(* CODESYS project mqtt.sharememory.gps.20211124.1.project

Project tree, tasks and I/O mapping:
  Device : Changsha Xiangji-ARM Cortex A9(xilinx zynq7000)-linux, Changsha Xiangji Hiden Technology Co.Ltd, version 3.5.10.40
    application Application
      libraries: Standard, * (System); SysShm, * (System); SysTypes2 Interfaces, * (System); CAA Types Extern, 3.5.13.0 (CAA Technical Workgroup); CAA Net Base Services, 3.5.15.0 (CAA Technical Workgroup); CAA Memory, 3.5.12.0 (CAA Technical Workgroup); SysFile, 3.5.15.0 (System); CAA SerialCom, 3.5.15.0 (CAA Technical Workgroup); MIC7001 base library, 1.11 (Cyber-MI.com); CAA DTUtil Extern, 3.5.12.0 (CAA Technical Workgroup)
      task Task_mqtt (cyclic, interval 200 ms, priority 19) calls prg_mqtt, prg_gps, prg_jt808
      global variables GVL
      data type ret_index
      MQTT_Client/
        Function Blocks/
          function block FB_CalculateRemainingLength [ST]
          function block FB_DecodeRemainingLength [ST]
          function block FB_MQTTClient [ST]: m_fill_subscribe_buf, m_fill_publish_buf, m_fill_connect_buf, rm_return, m_read_config
          function block FB_Random [ST]
        Structs/
          data type DUT_json
        Functions/
          function real_arr2string [ST]
          function MQTTPacket_encode [ST]
          function MQTTPacket_len [ST]
          function MQTT_connect_len [ST]
          function arr2json_model [ST]
          function json2arr [ST]
          function get_sub_string [ST]
          function count_char_in_string [ST]
          function rm_left [ST]
          function real2string [ST]
        program prg_mqtt [CFC]: ACT_boot, ACT_publish, ACT_recv_proc, ACT_first_buffer, ACT_normal_buffer, ACT_running_light, proc_get_command, proc_set_command, find_key
      gps/
        programs/
          program prg_gps [ST]
        Structs/
          data type stShmJT808Down
          data type stLocationExt
          data type stShmJT808Up
          data type stLocationBase
          data type stCanFrm
          data type nmeaTIME
          data type nmeaGPRMC
        functions/
          function nmea_parse_time [ST]
          function nmea_parse_date [ST]
          function get_latlon_from_str [ST]
          function nmea_parse_GPRMC [ST]
          function get_sub_string_1 [ST]
        functionblocks/
          function block Com_gps [ST]
      program prg_jt808 [ST]: send_to_server, read_from_server, init_shm
    SoftMotion General Axis Pool
  text list GlobalTextList
  5ce3da45-db07-42e7-a21c-a00fff4ed8f6|C:\Users\pengriguang\Desktop\cyber-tftp\huanweiche.bmp
*)

// Device/Application/ret_index
{attribute 'qualified_only'}
{attribute 'strict'}
TYPE ret_index :
(
	start := 0,
	cntr_box,
	cntr_lock,
	hours_e,
	fuel_work,
	fuel_idle
);
END_TYPE

// Device/Application/MQTT_Client/Structs/DUT_json
TYPE DUT_json :
STRUCT
	key:STRING(32);
	value_dint : DINT;
	value_real : REAL;
	value_str : STRING(256);
	val_tp : UINT;  //0:  int,   1: real,    2: string
END_STRUCT
END_TYPE

// Device/Application/gps/Structs/stShmJT808Down
TYPE stShmJT808Down :  // JT808下行数据
STRUCT
	location_interval:DINT;  // 位置信息发送间隔， 单位： ms
	ctrl : DINT;   // 车辆控制命令
END_STRUCT
END_TYPE

// Device/Application/gps/Structs/stLocationExt
TYPE stLocationExt :
STRUCT
	km_all: DINT;  // km all
	fuel:INT;   // fuel meter
	speed: INT;  // speed can
	lac:DINT; 
	cid:DINT;
	fuel_trip:DINT; // 本行程油耗
	fuel_all:DINT; 
	fuel_r_h:DINT;  // 0.05L/h
	fuel_r_l:DINT;  //  1/512Km/L
END_STRUCT
END_TYPE

// Device/Application/gps/Structs/stShmJT808Up
TYPE stShmJT808Up :   // 发送到服务器的上行数据
STRUCT
    location:stLocationBase;
	loc_ext:stLocationExt;
	can_data:stCanFrm;
END_STRUCT
END_TYPE

// Device/Application/gps/Structs/stLocationBase
TYPE stLocationBase :
STRUCT
	warning : UDINT;
    status : UDINT;
    latitude : DINT;
    longitude : DINT;
    altitude : INT;
    speed : INT;
    bearing : INT;
    asc_time :ARRAY[0..5] OF BYTE;  // ascii YYMMDDhhmmss (GMT+8)
END_STRUCT
END_TYPE

// Device/Application/gps/Structs/stCanFrm
TYPE stCanFrm :
STRUCT
	sn:UDINT;  // 每次更新内容后加一，用于通知底层发送程序
	id:UDINT;  //  CAN id
	data:ARRAY[0..7] OF BYTE;  // 8个字节 数据
END_STRUCT
END_TYPE

// Device/Application/gps/Structs/nmeaTIME
TYPE nmeaTIME :
STRUCT
	year:DINT;
	month:DINT;
	day:DINT;
	hour:DINT;
	minute:DINT;
	second:DINT;
	hsecond:DINT;
END_STRUCT
END_TYPE

// Device/Application/gps/Structs/nmeaGPRMC
TYPE nmeaGPRMC :
STRUCT
	utc : nmeaTIME;
	status : STRING(1);
	lat : REAL;
	ns : STRING(1);
	lon : REAL;
	ew : STRING(1);
	speed : REAL;
	direction : REAL;
	declination : REAL;
	declin_ew : STRING(1);
	mode : STRING(1);
END_STRUCT
END_TYPE

// Device/Application/GVL
{attribute 'qualified_only'}
VAR_GLOBAL PERSISTENT RETAIN
	ret_val1: DINT;  
	ret_val2: Dint;
END_VAR

VAR_GLOBAL CONSTANT
	TYPE_DINT:UINT := 0;
	TYPE_REAL:UINT := 1;
	TYPE_STRING:UINT := 2;
END_VAR

VAR_GLOBAL
	mqtt_interval : DINT := 5;  //mqtt package interval of publish to server
END_VAR

// Device/Application/MQTT_Client/prg_mqtt
PROGRAM prg_mqtt
VAR_INPUT
	mode_set :DINT := 99;
END_VAR
VAR
	FB_MQTTClient_0: FB_MQTTClient;
	
	//topic : STRING(255) := '/sys/a1SB8J9cA4L/CMI010319120011/thing/model/up_raw';
	//topic : STRING(255) := '/a1SB8J9cA4L/CMI010319120011/user/to_app';
	payload : STRING(255) := '{"RPM": 1234, "Hours": 2345}';
	
	//subscribe : STRING(255) := '/a1SB8J9cA4L/CMI010319120011/user/from_app';
	
	xPub : BOOL := FALSE;
	xSub : BOOL := FALSE;
	xBooted :BOOL := FALSE;
	
	ton_pub : ton;
	
	val_payload:ARRAY[0..32] OF dut_json;
	rpm_value : DINT := 1000;
	hours_value :REAL := 680;
	time_value : STRING;
	sn_value : STRING(128);
	lac_str:STRING(128);
	cid_str:STRING(128);
	press_value :REAL := 20.1;
	
	recv_data : ARRAY[0..32] OF DUT_json;
	old_recv_cntr:UDINT := 0;
	payload_len :INT;
	
	mqtt_first :BOOL := TRUE;
	ton_running:ton:=(pt := T#500MS);
	led_run:BOOL := FALSE;
	led_err:BOOL := FALSE;
	led_usr:BOOL := FALSE;
	pkg_id :DINT := 0;
	i :DINT;
	hour_today:REAL := 2.0;
	pub_cntr :DINT := 0;
	
	press:DWORD;
	oil :DWORD;
	temp : DWORD;
	send_serial:DINT := 0;  // 发送帧的序列号
	arr : ARRAY [0..19] OF REAL;
	
	angle:REAL := 60.0;
	length:REAL := 0.0;
END_VAR

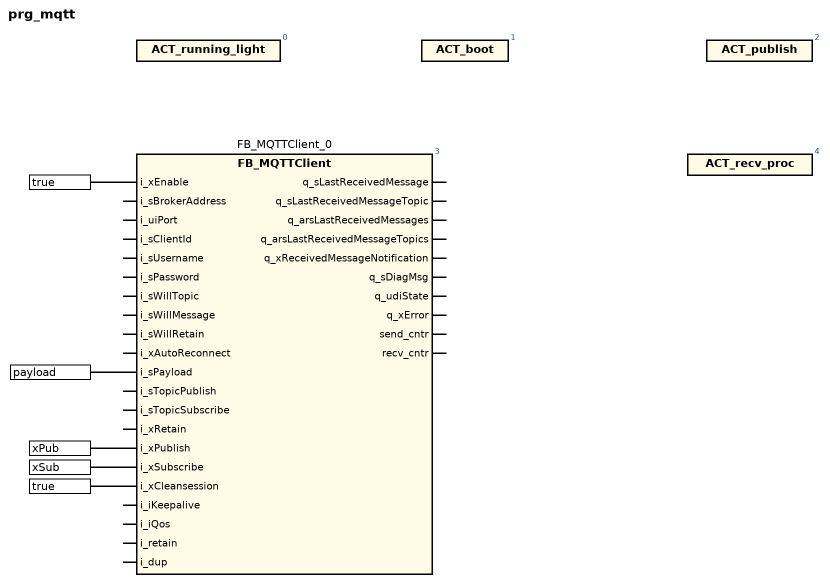
ACT_running_light();
ACT_boot();
ACT_publish();
FB_MQTTClient_0(
    i_xEnable := true,
    i_sPayload := payload,
    i_xPublish := xPub,
    i_xSubscribe := xSub,
    i_xCleansession := true); // FB_MQTTClient
ACT_recv_proc();

ACTION ACT_boot:
IF NOT xbooted THEN
	IF FB_MQTTClient_0.q_udiState = 60 THEN
		FB_MQTTClient_0.i_xSubscribe := TRUE;
		xBooted := TRUE;
	END_IF
END_IF
END_ACTION

ACTION ACT_publish:
IF FB_MQTTClient_0.q_udiState <> 60 THEN   //not ready, return and wait
	xPub := FALSE;
	RETURN;
END_IF

IF mqtt_first THEN
	mqtt_first := FALSE;
	ACT_first_buffer();
	xPub := TRUE;
	RETURN;
END_IF

ton_pub(in := NOT ton_pub.Q, pt := ANY_TO_TIME(gvl.mqtt_interval*1000));   // second to ms
IF ton_pub.Q THEN
	ACT_normal_buffer();
	xPub := TRUE;
ELSE
	xPub := FALSE;
END_IF
END_ACTION

ACTION ACT_recv_proc:
(*
	cmd:  	set, get          			//命令字, set:设置参数或者执行命令，  get：点播数据或参数
	act:  	lock, unlock, reboot		//动作类型
	grade:  1, 2, 3, 4					//动作级别
	delay:  0, 60, 3600					//延迟时间,单位： 秒
*)

IF old_recv_cntr = FB_MQTTClient_0.recv_cntr THEN  //no new message
	RETURN;
END_IF
old_recv_cntr := FB_MQTTClient_0.recv_cntr;

payload_len := json2arr(json := FB_MQTTClient_0.q_sLastReceivedMessage, pArr := ADR(recv_data), max_len := 32);
IF payload_len = 0 THEN
	RETURN;
END_IF

i := find_key(key := 'cmd');
IF i >= 0 AND recv_data[i].val_tp = GVL.TYPE_STRING THEN 
	IF  recv_data[i].value_str = 'get' THEN
		proc_get_command();
	ELSIF recv_data[i].value_str = 'set' THEN
		proc_set_command();
	END_IF
END_IF
END_ACTION

ACTION ACT_first_buffer:

val_payload[0].key := 'sn';
val_payload[0].val_tp := GVL.TYPE_STRING;
IF MIC7001_base.read_sn(ADR(sn_value)) THEN
	val_payload[0].value_str := sn_value;
ELSE
	val_payload[0].value_str := 'SN Error';
END_IF

val_payload[1].key := 'lac';
val_payload[1].val_tp := GVL.TYPE_STRING;

val_payload[2].key := 'cid';
val_payload[2].val_tp := GVL.TYPE_STRING;

IF MIC7001_base.read_location(lac := ADR(lac_str), ci := ADR(cid_str)) THEN
	val_payload[1].value_str := lac_str; 
	val_payload[2].value_str := cid_str; 
ELSE
	val_payload[1].value_str := 'lac_error'; 
	val_payload[2].value_str := 'cid_error'; 
END_IF

payload := arr2json_model(arr := val_payload, num := 3);
END_ACTION

ACTION ACT_normal_buffer:
// 数据太多，分帧发送  0~3 共4帧， 可以把需要同时发送的关联数据放在一帧中
CASE send_serial OF
0:	
	val_payload[0].key := 'BoxNo';
	val_payload[0].val_tp := GVL.TYPE_STRING; 
	val_payload[0].value_str := 'Box123456'; 

	val_payload[1].key := 'digi_0_29';
	val_payload[1].val_tp := GVL.TYPE_DINT; 
	val_payload[1].value_dint.0 := TRUE; //bForward;   // 前进档
	val_payload[1].value_dint.1 := FALSE; //bBackward;   // 前进档
	// ...
	val_payload[1].value_dint.29 := TRUE;  // bLocked;   // 属具已闭锁
	
	
	val_payload[2].key := 'digi_30_59';
	val_payload[2].val_tp := GVL.TYPE_DINT; 
	val_payload[2].value_dint := 12345;

	val_payload[3].key := 'digi_60_89';
	val_payload[3].val_tp := GVL.TYPE_DINT; 
	val_payload[3].value_dint := 12345; 

	val_payload[4].key := 'digi_90_119';
	val_payload[4].val_tp := GVL.TYPE_DINT; 
	val_payload[4].value_dint := 12345;  	
(*  ana_0_19	
0 发动机转速
1 发动机水温
2 发动机机油压力
3 发动机燃油箱体积
4 变速箱涡轮转速
5 变速箱温度
6 变速箱压力
7 吊载重量
8 前伸距
9 臂架角度
10 臂架长度
11 刹车油温度
12 液压油温度
13 俯仰动作手柄输入
14 伸缩动作手柄输入
15 吊具旋转动作输入
16 吊具侧移动作输入
17 整机故障代码
*)
	val_payload[5].key := 'ana_0_19';
	val_payload[5].val_tp := GVL.TYPE_STRING;
    arr[0] := 123; // gvl.rpm;
    arr[1] := 345.5678; // gvl.temp;
    arr[2] := 888; // gvl.press;t
	
	arr[8] := 4.2;   // 前伸距离 
	arr[9] := angle;   // 臂架角度
	arr[10] := length;   // 臂架长度
	
	angle := 60;
	
	length := length + 0.3;
	IF length > 7.2 THEN
		length := 0;
	END_IF
	
	// ...
    arr[17] := 16#01020304; // gvl.errorcode
	val_payload[5].value_str := real_arr2string(arr, 18); 
	
	payload := arr2json_model(arr := val_payload, num := 6);
	
1:
	val_payload[0].key := 'BoxNo';
	val_payload[0].val_tp := GVL.TYPE_STRING; 
	val_payload[0].value_str := 'Box123456'; 

	val_payload[1].key := 'digi_0_29';
	val_payload[1].val_tp := GVL.TYPE_DINT; 
	val_payload[1].value_dint := 12345; 
	
	val_payload[2].key := 'digi_30_59';
	val_payload[2].val_tp := GVL.TYPE_DINT; 
	val_payload[2].value_dint := 12345;

	val_payload[3].key := 'digi_60_89';
	val_payload[3].val_tp := GVL.TYPE_DINT; 
	val_payload[3].value_dint := 12345; 

	val_payload[4].key := 'digi_90_119';
	val_payload[4].val_tp := GVL.TYPE_DINT; 
	val_payload[4].value_dint := 12345;  
(*  ana_20_39
0 吊箱总数
1 旋锁计数
2 伸出PWM值
3 缩回PWM值
4 仰起PWM值
5 俯下PWM值
6 正面吊左无杆腔压力
7 正面吊右有杆腔压力
8 正面吊右无杆腔压力
9 正面吊伸缩压力
10 设备行驶速度
11 液压系统压力
12 力矩百分比
*)	
	val_payload[5].key := 'ana_20_39';
	val_payload[5].val_tp := GVL.TYPE_STRING;
    arr[0] := 333; // gvl.box_all;
    arr[1] := 555; // gvl.lock_all;
    arr[2] := 1357; // gvl.pwm_out;
	// ...
    arr[12] := 82; // gvl.tor
	val_payload[5].value_str := real_arr2string(arr, 13); 
	
	payload := arr2json_model(arr := val_payload, num := 6);
2:
	val_payload[0].key := 'BoxNo';
	val_payload[0].val_tp := GVL.TYPE_STRING; 
	val_payload[0].value_str := 'Box123456'; 

	val_payload[1].key := 'digi_0_29';
	val_payload[1].val_tp := GVL.TYPE_DINT; 
	val_payload[1].value_dint := 12345; 
	
	val_payload[2].key := 'digi_30_59';
	val_payload[2].val_tp := GVL.TYPE_DINT; 
	val_payload[2].value_dint := 12345;

	val_payload[3].key := 'digi_60_89';
	val_payload[3].val_tp := GVL.TYPE_DINT; 
	val_payload[3].value_dint := 12345; 

	val_payload[4].key := 'digi_90_119';
	val_payload[4].val_tp := GVL.TYPE_DINT; 
	val_payload[4].value_dint := 12345;  
(*  ana_40_59
0 发动机运行时间
1 发动机故障SPN码
2 发动机后处理SPN码
3 发动机蓄电池电压
4 总油耗
5 工作油耗
6 怠速油耗
7 发动机瞬时油耗
8 发动机怠速工作时长
9 刹车踏板制动百分比
10 油门踏板百分比
11 变速箱SPN_L
12 变速箱SPN_H
13 左前轮胎外侧胎压
14 左前轮胎内侧胎压
15 右前轮胎外侧胎压
16 右前轮胎内侧胎压
17 左后轮胎胎压
18 右后轮胎胎压
*)	
	val_payload[5].key := 'ana_40_59';
	val_payload[5].val_tp := GVL.TYPE_STRING;
    arr[0] := 333; // 
    arr[1] := 555; // 
    arr[2] := 1357; // 
	arr[3] := 28.1;
	arr[4] := 12345.6;
	arr[5] := 10000;
	arr[6] := 2345.6;
	arr[7] := 2.6;
	// ...
	arr[17] := 2.7;
	arr[18] := 2.9;
	val_payload[5].value_str := real_arr2string(arr, 19); 
	
	payload := arr2json_model(arr := val_payload, num := 6);

3:
	val_payload[0].key := 'BoxNo';
	val_payload[0].val_tp := GVL.TYPE_STRING; 
	val_payload[0].value_str := 'Box123456'; 

	val_payload[1].key := 'digi_0_29';
	val_payload[1].val_tp := GVL.TYPE_DINT; 
	val_payload[1].value_dint := 12345; 
	
	val_payload[2].key := 'digi_30_59';
	val_payload[2].val_tp := GVL.TYPE_DINT; 
	val_payload[2].value_dint := 12345;

	val_payload[3].key := 'digi_60_89';
	val_payload[3].val_tp := GVL.TYPE_DINT; 
	val_payload[3].value_dint := 12345; 

	val_payload[4].key := 'digi_90_119';
	val_payload[4].val_tp := GVL.TYPE_DINT; 
	val_payload[4].value_dint := 12345;  
(*  ana_20_39
设备类型
生产年份
车号
设备品牌
发动机类型
变速箱类型
驱动桥类型
吊具类型
吊具程序版本号
主机程序版本号
吊重箱数量
*)	
	val_payload[5].key := 'ana_60_79';
	val_payload[5].val_tp := GVL.TYPE_STRING;
    arr[0] := 333; // gvl.
    arr[1] := 555; // gvl.
    arr[2] := 1357; // gvl.
	// ...
    arr[10] := 82; // gvl.
	val_payload[5].value_str := real_arr2string(arr, 11); 
	
	payload := arr2json_model(arr := val_payload, num := 6);
4:
	val_payload[0].key := 'BoxNo';
	val_payload[0].val_tp := GVL.TYPE_STRING; 
	val_payload[0].value_str := 'Box123456'; 

	val_payload[1].key := 'digi_0_29';
	val_payload[1].val_tp := GVL.TYPE_DINT; 
	val_payload[1].value_dint := 12345; 
	
	val_payload[2].key := 'digi_30_59';
	val_payload[2].val_tp := GVL.TYPE_DINT; 
	val_payload[2].value_dint := 12345;

	val_payload[3].key := 'digi_60_89';
	val_payload[3].val_tp := GVL.TYPE_DINT; 
	val_payload[3].value_dint := 12345; 

	val_payload[4].key := 'digi_90_119';
	val_payload[4].val_tp := GVL.TYPE_DINT; 
	val_payload[4].value_dint := 12345;  
	
(*  ana_80_99
锂电池SOC
。。。
。。。
*)	
	val_payload[5].key := 'ana_80_99';
	val_payload[5].val_tp := GVL.TYPE_STRING;
    arr[0] := 333; // gvl.
    arr[1] := 555; // gvl.
    arr[2] := 1357; // gvl.
	// ...
    arr[10] := 82; // gvl.
    arr[11] := 12; // gvl.
	
IF prg_gps.packGPRMC.status = 'A' THEN  // GPS定位成功
	arr[12] := prg_gps.packGPRMC.lat*1000000;    //维度 * 1000000
	arr[13] := prg_gps.packGPRMC.lon*1000000;	 //经度 * 1000000
END_IF
	val_payload[5].value_str := real_arr2string(arr, 14);
	
	payload := arr2json_model(arr := val_payload, num := 6);	
	
END_CASE


send_serial := send_serial + 1;
IF send_serial > 4 THEN
	send_serial := 0;
END_IF
END_ACTION

ACTION ACT_running_light:
ton_running(in := NOT ton_running.Q);
IF ton_running.Q THEN
	led_run := NOT led_run;
	led_usr := FALSE;
END_IF

IF FB_MQTTClient_0.q_udiState <> 60 THEN
	led_usr := TRUE;
END_IF
END_ACTION

ACTION proc_get_command:
(*
	cmd:  	get  	//命令字, get：点播数据或参数
	rpm:  	15		//点播转速， 上传15次
	press:  0		//点播压力， 持续上传
	fuel_all: 1	  	//点播总油耗，上传一次 					
*)
END_ACTION

ACTION proc_set_command:
(*
	cmd:  	set  	          	//命令字, set:设置参数或者执行命令，  get：点播数据或参数
	interval:	15				//设置上传间隔： 15秒
	act:  	lock, unlock		//锁机动作类型
	grade:  1, 2, 3, 4			//动作级别
	delay:  0, 60, 3600			//延迟时间,单位： 秒
*)

// check lock command 
i := find_key(key := 'act');
IF i >= 0 AND recv_data[i].val_tp = GVL.TYPE_STRING  THEN
  //
END_IF
END_ACTION

METHOD find_key : dint
VAR_INPUT
	key :STRING(32);
END_VAR
VAR
	i :UINT;
END_VAR
find_key := -1;

FOR i := 0 TO payload_len-1 DO
	IF key = recv_data[i].key THEN
		find_key := i;
		RETURN;
	END_IF
END_FOR

RETURN; // not find,  return -1
END_METHOD

END_PROGRAM

// Device/Application/MQTT_Client/Function Blocks/FB_MQTTClient
(*  mqtt client for MIC7001
    by zhoujihui@gmail.com
*)
FUNCTION_BLOCK FB_MQTTClient
VAR_INPUT
	// Enables the Function block, The rising Edge of this Input automatically connects to the MQTT Broker - Standard: TRUE
	i_xEnable: BOOL := TRUE;
	// IP-Address (example: 192.168.178.101) or Webaddress (www.mqtt-dashboard.com) of the MQTT-Broker
	i_sBrokerAddress: STRING(255) := '47.107.240.29';
	// Port of the MQTT-Broker - Standard: 1883
	i_uiPort: UINT := 1883;
	// clientId
	i_sClientId: STRING(255) := 'MIC7001 client Id';
	// Optional Username if required
	i_sUsername: STRING(255) := '';
	// Optional Password if required
	i_sPassword: STRING(255) := '';
	// Last Will Topic if required (Automatically enables Will Message if changed) - otherwise leave untouched
	i_sWillTopic: STRING(255) := '';
	// Last Will Message if required - otherwise leave untouched
	i_sWillMessage: STRING(255) := '';
	// Retain Last Will Message, if required Standard: FALSE - otherwise leave untouched 
	i_sWillRetain: BOOL := FALSE;	
	// Automatically try to reconnect after an Exception - Standard: TRUE
	i_xAutoReconnect: BOOL := TRUE;
	// PayLoad to Publish
	i_sPayload: STRING(255) := '';
	// Topic to Publish to
	i_sTopicPublish: STRING(255) := '/MIC7001/without/config/files';
	// Topic to Subscribe
	i_sTopicSubscribe: STRING(255) := '';
	// Retain Flag Forces the Broker to Retain the Last Mesage - Standard: TRUE
	i_xRetain: BOOL := TRUE;
	// Publish the Payload to the Topic of the MQTT-Broker
	i_xPublish: BOOL:=FALSE;
	// Subscribe to the Topic given to the Input i_sTopicSubscribe
	i_xSubscribe: BOOL:=FALSE;
	// clean session
	i_xCleansession : BOOL := FALSE;
	// keep alive
	i_iKeepalive :INT := 60000;
	// QoS of publish packet
	i_iQos : BYTE := 0;
	// retain
	i_retain : BOOL := FALSE;
	// dup
	i_dup :BOOL := FALSE;
	
END_VAR
VAR_OUTPUT
	// Message Received from a subsribed Topic
	q_sLastReceivedMessage: STRING(255);
	// Topic Message Received
	q_sLastReceivedMessageTopic: STRING(255);	
	// Last 25 Received Messages
	q_arsLastReceivedMessages: STRING(255);
	// Last 25 Topics Received
	q_arsLastReceivedMessageTopics: STRING(255);	
	// Message Received Notification
	q_xReceivedMessageNotification: BOOL;
	// Diag Message
	q_sDiagMsg: STRING(255);
	// Current State of the Function Block
	q_udiState: UDINT;
	// Error Flag
	q_xError: BOOL;
	//publish message counter
	send_cntr :UDINT := 0;
	//received message counter
	recv_cntr: UDINT := 0;
END_VAR
VAR
	R_TRIG_Enable: R_TRIG;

	diResult: CAA.SIZE;
	IFB_CalculateRemainingLength: FB_CalculateRemainingLength;
	IFB_Random: ARRAY[0..9] OF FB_Random;
	wKeepAlive: WORD := 0;
	IoCtlParameter : DINT := 1;

	R_TRIG_Publish: R_TRIG;
	R_TRIG_Subscribe: R_TRIG;

	uiYear:UINT;
	uiMonth: UINT;
	uiDay: UINT;
	uiHour: UINT;
	uiMinute: UINT;
	uiSecond: UINT;
	
	TON_TimeOut: ton;
	wTimeOutValue: WORD;
	udiLastState: UDINT;
	
	xResultDisconnect: BOOL;
	QI: INT;
	
	iIndexCount: INT;
	wPacketIdentifierCount: WORD :=0;
	uiPayLoadLength: uint;
	
	xPublish: BOOL;
	xSubscribe: BOOL;
	
	i: INT;

	hSock:RTS_IEC_HANDLE;
	pSock_create_rst: POINTER TO RTS_IEC_RESULT;
	pSock_recv_rst: POINTER TO RTS_IEC_RESULT;
	pSock_send_rst: POINTER TO RTS_IEC_RESULT;

	ui_rc_disconnect : UDINT;
	pInaddr:POINTER TO STRING;
	
	tcp_client : NBS.TCP_Client;
	tcp_connection : CAA.HANDLE;
	tcp_send : NBS.TCP_Write;
	tcp_recv : NBS.TCP_Read;
	s_send_buf : ARRAY[0..999] OF BYTE;
	s_recv_buf : ARRAY[0..999] OF BYTE;
	udi_time_out : UDINT;
	server_ip : NBS.IP_ADDR;
	buf_size : CAA.size;
	recv_len : INT;

	header :BYTE ; 
	bytes_len_rem : INT;
	length_topic : INT;
	recv_qos : BYTE := 0;
	id_msb : BYTE;
	id_lsb : BYTE;
	hFile: RTS_IEC_HANDLE;
	udiOpenError: RTS_IEC_RESULT;
	udiReadError: RTS_IEC_RESULT;
	str_size: __XWORD;
	udiByteRead: LWORD;	
	str_temp:STRING(255);
	error_cntr : DINT := 0;
END_VAR


R_TRIG_Enable(CLK:=i_xEnable);
R_TRIG_Publish(CLK:=i_xPublish);
R_TRIG_Subscribe(CLK:=i_xSubscribe);

IF (R_TRIG_Publish.Q) THEN
	xPublish:=TRUE;
END_IF

IF (R_TRIG_Subscribe.Q) THEN
	xSubscribe:=TRUE;
END_IF

CASE q_udiState OF
//0: Wait for Enable
0: 	wTimeOutValue:=0;
	
	IF (NOT q_xError) THEN	
		q_sDiagMsg:='Wait for Enable';
	END_IF
	
	IF (i_xEnable OR (i_xAutoReconnect AND q_xError)) THEN
		IF m_read_config() THEN
			q_xError := FALSE;
			q_udiState:=5;
			tcp_client(xEnable := FALSE);
			server_ip.sAddr := i_sBrokerAddress;
			tcp_client.xEnable := TRUE;			
			q_sDiagMsg:='Creating TCP connect';
		ELSE
			q_xError := TRUE;
			q_sDiagMsg:='Failed reading config files';
			q_udiState:=99;
		END_IF
		
	END_IF

5:  
	IF tcp_client.xActive THEN
		q_udiState := 15;
		q_sDiagMsg:='Initialize send-Buffer';
	END_IF
	
	wTimeOutValue:=3000;
	IF (TON_TimeOut.Q) THEN
		q_udiState:=0;	
	END_IF		

//15: Initialize OutBuffer
15:
	buf_size := m_fill_connect_buf();
	IF buf_size > 0 THEN
		tcp_send.szSize := buf_size; 
		tcp_send(xExecute := FALSE);
		tcp_send.xExecute := TRUE;
		tcp_recv.xEnable := TRUE;
		
		q_udiState:=20;
		q_sDiagMsg:='Connect to MQTT-Broker';
	ELSE
		q_xError := TRUE;
		q_sDiagMsg:='Send buffer is Error.';
		q_udiState:=0;
	END_IF
	
//20: Send Connect	
20:		
	wTimeOutValue:=1000;
	tcp_recv(hConnection := tcp_connection, szSize := 1024, pData := ADR(s_recv_buf));
	IF tcp_recv.xReady  THEN
		q_udiState:= 30;
	END_IF
	
	IF (TON_TimeOut.Q) THEN
		q_udiState:=0;	
		q_xError := TRUE;
		q_sDiagMsg:='Connecting to MQTT-Broker (MQTT Control Packet) Timed out';
	END_IF
//30: Analyze CONNACK
30:	q_sDiagMsg:='Analyze connack';
	wTimeOutValue:=0;
	
	IF (s_recv_buf[0] = 32 AND s_recv_buf[3] = 0) THEN
		q_udiState := 60;
	ELSE
		//Return code repsone (2nd Byte): 
		//0: Connection Accepted
		//1: Connection Refused, unacceptable protocol version
		IF (s_recv_buf[3] = 1) THEN
			q_sDiagMsg:='Connection Refused, unacceptable protocol version';
		END_IF
		//2: Connection Refused, identifier rejected
		IF (s_recv_buf[3] = 2) THEN
			q_sDiagMsg:='Connection Refused, identifier rejected';
		END_IF
		//3: Connection Refused, Server unavailable
		IF (s_recv_buf[3] = 3) THEN
			q_sDiagMsg:='Connection Refused, Server unavailable';
		END_IF		
		//4: Connection Refused, bad Username or passworrd
		IF (s_recv_buf[3] = 4) THEN
			q_sDiagMsg:='Connection Refused, bad Username or password';
		END_IF	
		//5: Connection Refused, not autorized
		IF (s_recv_buf[3] = 5) THEN
			q_sDiagMsg:='Connection Refused, not autorized';
		END_IF	
		q_xError := TRUE;
		q_udiState := 90;	
	END_IF
	
//60: Wait for Publish or Disconnect (Enable low)
60:	q_sDiagMsg:='Wait for Publish or Subscribe or Disconnect (Enable low)';
	wTimeOutValue:=0;
	q_xReceivedMessageNotification:= FALSE;

	IF (xPublish) THEN
		xPublish:=FALSE;
		q_udiState := 70;	
	END_IF
	IF (xSubscribe) THEN
		xSubscribe:=FALSE;
		q_udiState := 65;	
	END_IF
	IF (NOT i_xEnable) THEN
		q_udiState := 80;	
	END_IF
	
	tcp_recv(hConnection := tcp_connection, szSize := 1024, pData := ADR(s_recv_buf));
	IF tcp_recv.szCount > 2 THEN
		header := s_recv_buf[0];
		IF header.5 AND header.4 AND tcp_recv.szCount < 1024 THEN   // publish:  0x30
			q_xReceivedMessageNotification:= TRUE;
			diResult := tcp_recv.szCount;
			q_udiState := 63;
			
		END_IF	
	END_IF
	
//Analyze Publish Message from Broker
63: q_sDiagMsg:='Analyze Publish Message from Broker';
	wTimeOutValue:=0;

	IFB_CalculateRemainingLength(wNumberOfBytes:=ANY_TO_WORD(diResult-2));
	bytes_len_rem := IFB_CalculateRemainingLength.iNumberOfBytesRemianingLengthField;
	length_topic := BYTE_TO_INT(s_recv_buf[bytes_len_rem+1])*256 + s_recv_buf[bytes_len_rem+2];
	IF length_topic > 128 THEN
		q_udiState := 60;
		RETURN;	
	END_IF
	
	uiPayLoadLength:=ANY_TO_UINT(diResult - length_topic - 1 - bytes_len_rem - 2);
	header := s_recv_buf[0];
	
	recv_qos := 0;
	IF header.1 OR header.2 THEN //Qos > 0
		uiPayLoadLength :=  uiPayLoadLength - 2;  //remove 2bytes of packet Id
		IF header.1 THEN
			recv_qos := 1;
		ELSIF header.2 THEN
			recv_qos := 2;
		END_IF	

		id_msb := s_recv_buf[1+bytes_len_rem + 2 + length_topic];
		id_lsb := s_recv_buf[1+bytes_len_rem + 2 + length_topic+1];
	END_IF
	
	mem.MemFill(ADR(q_sLastReceivedMessage),255,0);
	mem.MemFill(ADR(q_sLastReceivedMessageTopic),255,0);
	MEM.MemMove(ADR(s_recv_buf[diResult-uiPayLoadLength]),ADR(q_sLastReceivedMessage),uiPayLoadLength);
	MEM.MemMove(ADR(s_recv_buf[IFB_CalculateRemainingLength.iNumberOfBytesRemianingLengthField+3]),ADR(q_sLastReceivedMessageTopic),length_topic);
	
	q_arsLastReceivedMessageTopics:=q_sLastReceivedMessageTopic;
	q_arsLastReceivedMessages:=q_sLastReceivedMessage;
	
	diResult:=0;
	recv_cntr := recv_cntr + 1;
	IF recv_qos = 0 THEN
		q_udiState := 60;
	ELSIF recv_qos = 1 THEN
		
		s_send_buf[0] := 16#40;  //type: puback
		s_send_buf[1] := 2;
		s_send_buf[2] := id_msb;
		s_send_buf[3] := id_lsb;
		tcp_send(xExecute := FALSE);
		tcp_send.xExecute := TRUE;
		tcp_send.szSize := 4;
		q_udiState := 64; // send ack
		wTimeOutValue:=1000;
		q_sDiagMsg:='Send ack to broker';
	ELSE  // qos = 2, not support yet
		q_udiState := 60;
	END_IF	

64:
	IF tcp_send.xDone THEN
		q_udistate := 60;
	END_IF
//65: Subscribe to Topic
65: q_sDiagMsg:='Subscribe to Topic';
	wTimeOutValue:=1000;
	
	buf_size := m_fill_subscribe_buf();
	IF buf_size > 0 THEN
		tcp_send.szSize := buf_size; 
		tcp_send(xExecute := FALSE);
		tcp_send.xExecute := TRUE;
		tcp_recv.xEnable := TRUE;
		q_udiState:=66;	
	ELSE
		q_xError := TRUE;
		q_sDiagMsg:='Subscribe buffer is Error.';
		q_udiState:=0;
	END_IF
	
	tcp_recv(hConnection := tcp_connection, szSize := 1024, pData := ADR(s_recv_buf));
	IF tcp_recv.xDone THEN 
		q_udiState:=66;	
	END_IF	
	IF (TON_TimeOut.Q) THEN
		q_udiState:=90;	
		q_xError := TRUE;
		q_sDiagMsg:='Subscribe (MQTT Control Packet) Timed out';
	END_IF	
	
//66: Wait for SUBACK from Broker
66: //diResult := SysSockRecv(hSocket := hSock,pbyBuffer:=ADR(inBuffer),diBufferSize:=500,diFlags:=0, ADR(pSock_recv_rst));
	q_sDiagMsg:='Wait for SUBACK from Broker';
	wTimeOutValue:=1000;
	tcp_recv(hConnection := tcp_connection, szSize := 1024, pData := ADR(s_recv_buf));
	IF tcp_recv.szCount > 0 THEN
		q_udiState:=67;	
		diResult:=0;
	END_IF
	IF (TON_TimeOut.Q) THEN
		q_udiState:=90;	
		q_xError := TRUE;
		q_sDiagMsg:='Waiting for "Suback" from MQTT-Broker Timed out';
	END_IF

//67: Analyze SUBACK
67:	q_sDiagMsg:='Analyze SUBACK';
	wTimeOutValue:=0;
	tcp_recv(hConnection := tcp_connection, szSize := 1024, pData := ADR(s_recv_buf));
	recv_len := ANY_TO_INT(tcp_recv.szCount);
	IF (s_recv_buf[recv_len-1] < 16#80) THEN
		q_udiState := 60;
		diResult:=0;
	ELSE	
		q_udiState:=90;	
		q_xError := TRUE;
		q_sDiagMsg:='Suback Message reported Failure (Return code 0x80)';
	END_IF
	
//70: Publish Message
70: 
	buf_size := m_fill_publish_buf();

	IF buf_size > 0 THEN
		tcp_send.szSize := buf_size; 
		tcp_send(xExecute := FALSE);
		tcp_send.xExecute := TRUE;
		tcp_recv.xEnable := TRUE;
		q_sDiagMsg:='Publish Message';
		wTimeOutValue:=1000;		
		q_udiState:=75;	
	END_IF
	
75:	
	IF (tcp_send.xDone > 0) THEN 
		q_udiState:=60;	
		send_cntr := send_cntr + 1;
	END_IF	
	IF (TON_TimeOut.Q) THEN
		q_udiState:=90;	
		q_xError := TRUE;
		q_sDiagMsg:='Publishing Message (MQTT Control Packet) Timed out';
	END_IF

//80: Send "Disconnect"
80: s_send_buf[0] := 224;		//MQTT Control Packet Type
	s_send_buf[1] := 0;			//Remaining Length (0)
	tcp_send.szSize := 2;
	tcp_send(xExecute := FALSE);
	tcp_send.xExecute := TRUE;
	
	q_sDiagMsg:='Send Disconnect notification to server';
	wTimeOutValue:=1000;
	q_udiState:=85;

85:	
	IF (tcp_send.xDone) THEN 
		diResult:=0;
		q_udiState:=90;	
	END_IF	
	IF (TON_TimeOut.Q) THEN
		q_udiState:=90;	
		q_xError := TRUE;
		q_sDiagMsg:='Sending Disconnect to MQTT-Broker Timed out';
	END_IF	

//90: Disconnect Socket
90:	tcp_client.xEnable := FALSE;
	IF (NOT q_xError) THEN
		q_sDiagMsg:='Close TCP Socket';
	END_IF
	wTimeOutValue:=1000;
	IF (ui_rc_disconnect = 0) THEN 
		q_udiState:=0;	
	END_IF	
	IF (TON_TimeOut.Q) THEN
		q_udiState:=0;	
		q_xError := TRUE;
		q_sDiagMsg:='Closing TCP-Socket  Timed out';
	END_IF	

99: //error
	wTimeOutValue:=5000;
	IF (TON_TimeOut.Q) THEN
		q_udiState:=0;	
		q_xError := TRUE;
		q_sDiagMsg:='Error status Timed out';
	END_IF	
END_CASE

TON_TimeOut(IN:=(udiLastState=q_udiState) AND (wTimeOutValue <> 0) ,PT:=WORD_TO_TIME(wTimeOutValue));
udiLastState:=q_udiState;

IF q_udiState >= 5 THEN
	tcp_client(xEnable := TRUE, ipAddr := server_ip, uiPort := i_uiPort , udiTimeOut := 0, hConnection => tcp_connection);
	IF tcp_connection > 0 THEN
		tcp_send(udiTimeOut := udi_time_out, hConnection := tcp_connection, pData := ADR(s_send_buf));
	END_IF
END_IF

METHOD m_fill_subscribe_buf : CAA.SIZE
VAR_INPUT
END_VAR

VAR
	i : INT;
	ui_subscribe_len:INT;
	ui_mqtt_msg_len:INT;
	ptr : INT := 0;
	rem_len :INT := 0;
	packet_len : CAA.SIZE := 0;
	rc :INT := 0;
	
	flag :BYTE := 0;
END_VAR
m_fill_subscribe_buf := 0;

ui_subscribe_len := (LEN(i_sTopicSubscribe));

rem_len := ui_subscribe_len + 2 + 2 + 1;  //packet id: 2bytes,  length: 2bytes, QoS: 1byte 
packet_len := MQTTPacket_len(rem_len);

IF packet_len > SIZEOF(s_send_buf) THEN
	m_fill_subscribe_buf := 0;
	RETURN;
END_IF

ptr := 0;
// Header Flag. subscribe command.
flag := 16#82;

IF i_dup THEN
	flag := flag + 8;
END_IF

s_send_buf[ptr] := flag;  ptr := ptr + 1;

// Msg Len.
rc := MQTTPacket_encode(ADR(s_send_buf[ptr]), rem_len);   ptr := ptr + rc;

wPacketIdentifierCount:=wPacketIdentifierCount + 1;
IF (wPacketIdentifierCount = 0) THEN
	wPacketIdentifierCount:=1;
END_IF

// packet id	
s_send_buf[ptr] := UINT_TO_BYTE(wPacketIdentifierCount / 256); ptr := ptr + 1;
s_send_buf[ptr] := UINT_TO_BYTE(wPacketIdentifierCount MOD 256); ptr := ptr + 1;

// topic Length.
s_send_buf[ptr] := UINT_TO_BYTE(ui_subscribe_len / 256); ptr := ptr + 1;
s_send_buf[ptr] := UINT_TO_BYTE(ui_subscribe_len MOD 256); ptr := ptr + 1;

//topic subscribe
FOR i:=0 TO ui_subscribe_len-1 DO
	s_send_buf[ptr] := i_sTopicsubscribe[i]; ptr := ptr + 1;
END_FOR	

s_send_buf[ptr] := i_iQos;

m_fill_subscribe_buf := packet_len;
END_METHOD

METHOD m_fill_publish_buf : CAA.SIZE
VAR_INPUT
END_VAR

VAR
	i : INT;
	ui_client_id_len : INT;
	ui_topic_len :INT;
	ui_payload_len:INT;
	ui_mqtt_msg_len:INT;
	ptr : INT := 0;
	rem_len :INT := 0;
	packet_len : CAA.size := 0;
	rc :INT := 0;
	packet_id : UINT := 1;
	flag :BYTE := 0;
END_VAR
m_fill_publish_buf := 0;

ui_topic_len := (LEN(i_sTopicPublish));
ui_payload_len := (LEN(i_sPayload));

rem_len := ui_topic_len + 2 + ui_payload_len;
IF i_iQos > 0 THEN
	rem_len := rem_len + 2;  // add 2 bytes packet Id
END_IF

packet_len := MQTTPacket_len(rem_len);

IF packet_len > SIZEOF(s_send_buf) THEN
	m_fill_publish_buf := 0;
	RETURN;
END_IF

ptr := 0;
// Header Flag. Publish command.
flag := 16#30;  //publish
IF i_retain THEN
	flag := flag + 1;
END_IF

IF i_iQos > 0 AND i_iQos < 3 THEN
	flag := flag + i_iQos*2;
ELSE
	i_dup := 0;
END_IF

IF i_dup THEN
	flag := flag + 8;
END_IF

s_send_buf[ptr] := flag;  ptr := ptr + 1;

// Msg Len.
rc := MQTTPacket_encode(ADR(s_send_buf[ptr]), rem_len);   ptr := ptr + rc;

//topic
IF ui_topic_len > 0 THEN
	// topic Length.
	s_send_buf[ptr] := UINT_TO_BYTE(ui_topic_len / 256); ptr := ptr + 1;
	s_send_buf[ptr] := UINT_TO_BYTE(ui_topic_len MOD 256); ptr := ptr + 1;
	
	// topic
	FOR i:=0 TO ui_topic_len-1 DO
		s_send_buf[ptr] := i_sTopicPublish[i]; ptr := ptr + 1;
	END_FOR	
END_IF

IF i_iQos > 0 THEN
	wPacketIdentifierCount:=wPacketIdentifierCount + 1;
	IF (wPacketIdentifierCount = 0) THEN
		wPacketIdentifierCount:=1;
	END_IF
	s_send_buf[ptr] := UINT_TO_BYTE(wPacketIdentifierCount / 256); ptr := ptr + 1;
	s_send_buf[ptr] := UINT_TO_BYTE(wPacketIdentifierCount MOD 256); ptr := ptr + 1;
END_IF

//payload
IF ui_payload_len > 0 THEN
	// payload,  no length needed
	FOR i:=0 TO ui_payload_len-1 DO
		s_send_buf[ptr] := i_spayload[i]; ptr := ptr + 1;
	END_FOR	
END_IF

m_fill_publish_buf := packet_len;
END_METHOD

METHOD m_fill_connect_buf : CAA.SIZE
VAR_INPUT
END_VAR

VAR
	ui_client_id_len : INT;	
	ui_username_len : INT;
	ui_password_len : INT;
	ui_will_topic_len : INT;
	ui_will_msg_len : INT;
	ptr:INT := 0;  
	remaining_len :INT;
	packet_len :CAA.SIZE;
	rc :INT;
	flag : BYTE := 0;
END_VAR
m_fill_connect_buf := 0;

ui_client_id_len := (LEN(i_sclientid));
ui_username_len := (LEN(i_sUsername));
ui_password_len := (LEN(i_sPassword));
ui_will_topic_len := (len(i_sWillTopic));
ui_will_msg_len := (len(i_sWillMessage));

remaining_len := MQTT_connect_len(ui_client_id_len, ui_will_topic_len, ui_will_msg_len, ui_username_len, ui_password_len);
packet_len := MQTTPacket_len(remaining_len);

IF packet_len > SIZEOF(s_send_buf) THEN
	m_fill_connect_buf := 0;
	RETURN;
END_IF

ptr := 0;

// Header Flag. Connect command.
s_send_buf[ptr] := 16#10; ptr := ptr + 1;

// Msg Len.
rc := MQTTPacket_encode(ADR(s_send_buf[ptr]), remaining_len);   ptr := ptr + rc;


// Protocal Name Length.
s_send_buf[ptr] := 16#00; ptr := ptr + 1;
s_send_buf[ptr] := 16#04; ptr := ptr + 1;
// Protocal Name.
s_send_buf[ptr] := 16#4D; ptr := ptr + 1;
s_send_buf[ptr] := 16#51; ptr := ptr + 1;
s_send_buf[ptr] := 16#54; ptr := ptr + 1;
s_send_buf[ptr] := 16#54; ptr := ptr + 1;
// Version.
s_send_buf[ptr] := 16#04; ptr := ptr + 1;

// Connect Flags.
flag := 0;
IF i_xCleansession THEN
	flag := flag + 16#02;
END_IF

IF ui_username_len > 0 THEN
	flag := flag + 16#80;
END_IF

IF ui_password_len > 0 THEN
	flag := flag + 16#40;
END_IF

s_send_buf[ptr] := flag;  ptr := ptr + 1;

// Keep Alive.
s_send_buf[ptr] := INT_TO_BYTE(i_iKeepalive / 256); ptr := ptr + 1;
s_send_buf[ptr] := INT_TO_BYTE(i_iKeepalive MOD 256); ptr := ptr + 1;

// Client ID Length.
s_send_buf[ptr] := INT_TO_BYTE(ui_client_id_len / 256); ptr := ptr + 1;
s_send_buf[ptr] := INT_TO_BYTE(ui_client_id_len MOD 256); ptr := ptr + 1;
// Client ID.
FOR i:=0 TO ui_client_id_len-1 DO
	s_send_buf[ptr] := i_sClientId[i]; ptr := ptr + 1;
END_FOR

IF ui_will_topic_len > 0 THEN
	// will topic Length.
	s_send_buf[ptr] := INT_TO_BYTE(ui_will_topic_len / 256); ptr := ptr + 1;
	s_send_buf[ptr] := INT_TO_BYTE(ui_will_topic_len MOD 256); ptr := ptr + 1;
	// will topic.
	FOR i:=0 TO ui_will_topic_len-1 DO
		s_send_buf[ptr] := i_sWilltopic[i]; ptr := ptr + 1;
	END_FOR	
END_IF

IF ui_will_msg_len > 0 THEN
	// will message Length.
	s_send_buf[ptr] := INT_TO_BYTE(ui_will_msg_len / 256); ptr := ptr + 1;
	s_send_buf[ptr] := INT_TO_BYTE(ui_will_msg_len MOD 256); ptr := ptr + 1;
	// will message.
	FOR i:=0 TO ui_will_msg_len-1 DO
		s_send_buf[ptr] := i_sWillmessage[i]; ptr := ptr + 1;
	END_FOR	
END_IF

IF ui_username_len > 0 THEN
	// will message Length.
	s_send_buf[ptr] := INT_TO_BYTE(ui_username_len / 256); ptr := ptr + 1;
	s_send_buf[ptr] := INT_TO_BYTE(ui_username_len MOD 256); ptr := ptr + 1;
	// username
	FOR i:=0 TO ui_username_len-1 DO
		s_send_buf[ptr] := i_susername[i]; ptr := ptr + 1;
	END_FOR	
END_IF

IF ui_password_len > 0 THEN
	// will message Length.
	s_send_buf[ptr] := INT_TO_BYTE(ui_password_len / 256); ptr := ptr + 1;
	s_send_buf[ptr] := INT_TO_BYTE(ui_password_len MOD 256); ptr := ptr + 1;
	// password
	FOR i:=0 TO ui_password_len-1 DO
		s_send_buf[ptr] := i_spassword[i]; ptr := ptr + 1;
	END_FOR	
END_IF


m_fill_connect_buf := packet_len;
END_METHOD

METHOD PRIVATE rm_return : string(255)
VAR_INPUT
	str_in:STRING(255);
END_VAR

VAR
	str_rc:string(255);
	length:INT;
END_VAR
str_rc := str_in;

length := len(str_rc);
IF str_rc[length-1] = 10 THEN   // $N
	str_rc := left(str_rc, length-1);
END_IF

length := len(str_rc);
IF str_rc[length-1] = 10 THEN   // $N
	str_rc := left(str_rc, length-1);
END_IF

length := len(str_rc);
IF str_rc[length-1] = 10 THEN   // $N
	str_rc := left(str_rc, length-1);
END_IF

length := len(str_rc);
IF str_rc[length-1] = 10 THEN   // $N
	str_rc := left(str_rc, length-1);
END_IF

rm_return := str_rc;
END_METHOD

METHOD m_read_config : bool
VAR_INPUT
END_VAR
m_read_config := FALSE;

hFile := sysfileopen(szFile := '/userapp/mqtt_server.txt', am := sysfile.AM_READ, pResult:= ADR(udiOpenError));
IF hFile = RTS_INVALID_HANDLE THEN
	RETURN;
END_IF

//文件存在，开始读取内容
sysfile.SysFileSetPos(hFile:=hFile, ulOffset := 0);
FOR i := 0 TO 255 DO  str_temp[i] := 0; END_FOR
udiByteRead := sysfile.SysFileRead(hfile := hFile,pbyBuffer := ADR(str_temp), ulSize := 250, pResult := ADR(udiReadError));
str_temp := rm_return(str_temp);
IF udiByteRead > 7 THEN  
	i_sBrokerAddress := str_temp;
END_IF
sysfile.SysFileClose(hFile := hFile);	

hFile := sysfileopen(szFile := '/userapp/mqtt_port.txt', am := sysfile.AM_READ, pResult:= ADR(udiOpenError));
IF hFile = RTS_INVALID_HANDLE	THEN
	RETURN;
END_IF
 
//文件存在，开始读取内容
sysfile.SysFileSetPos(hFile:=hFile, ulOffset := 0);
FOR i := 0 TO 255 DO  str_temp[i] := 0; END_FOR
udiByteRead := sysfile.SysFileRead(hfile := hFile,pbyBuffer := ADR(str_temp), ulSize := 32, pResult := ADR(udiReadError));
str_temp := rm_return(str_temp);
IF udiByteRead > 2 THEN  
	i_uiPort := STRING_TO_UINT(str_temp);
END_IF
sysfile.SysFileClose(hFile := hFile);	

hFile := sysfileopen(szFile := '/userapp/mqtt_client_id.txt', am := sysfile.AM_READ, pResult:= ADR(udiOpenError));
IF hFile = RTS_INVALID_HANDLE	THEN
	RETURN;
END_IF 
//文件存在，开始读取内容
sysfile.SysFileSetPos(hFile:=hFile, ulOffset := 0);
FOR i := 0 TO 255 DO  str_temp[i] := 0; END_FOR
udiByteRead := sysfile.SysFileRead(hfile := hFile,pbyBuffer := ADR(str_temp), ulSize := 250, pResult := ADR(udiReadError));
str_temp := rm_return(str_temp);
IF udiByteRead > 7 THEN  
	i_sClientId := str_temp;
END_IF
sysfile.SysFileClose(hFile := hFile);	

hFile := sysfileopen(szFile := '/userapp/mqtt_username.txt', am := sysfile.AM_READ, pResult:= ADR(udiOpenError));
IF hFile = RTS_INVALID_HANDLE	THEN
	RETURN;
END_IF
 
//文件存在，开始读取内容
sysfile.SysFileSetPos(hFile:=hFile, ulOffset := 0);
FOR i := 0 TO 255 DO  str_temp[i] := 0; END_FOR
udiByteRead := sysfile.SysFileRead(hfile := hFile,pbyBuffer := ADR(str_temp), ulSize := 250, pResult := ADR(udiReadError));
str_temp := rm_return(str_temp);
IF udiByteRead > 7 THEN  
	i_sUsername := str_temp;
END_IF
sysfile.SysFileClose(hFile := hFile);	

hFile := sysfileopen(szFile := '/userapp/mqtt_password.txt', am := sysfile.AM_READ, pResult:= ADR(udiOpenError));
IF hFile = RTS_INVALID_HANDLE	THEN
	RETURN;
END_IF 
//文件存在，开始读取内容
sysfile.SysFileSetPos(hFile:=hFile, ulOffset := 0);
FOR i := 0 TO 255 DO  str_temp[i] := 0; END_FOR
udiByteRead := sysfile.SysFileRead(hfile := hFile,pbyBuffer := ADR(str_temp), ulSize := 250, pResult := ADR(udiReadError));
str_temp := rm_return(str_temp);
IF udiByteRead > 7 THEN
	i_sPassword := str_temp;
END_IF
sysfile.SysFileClose(hFile := hFile);	

hFile := sysfileopen(szFile := '/userapp/mqtt_topic_publish.txt', am := sysfile.AM_READ, pResult:= ADR(udiOpenError));
IF hFile = RTS_INVALID_HANDLE	THEN
	RETURN;
END_IF
 
//文件存在，开始读取内容
sysfile.SysFileSetPos(hFile:=hFile, ulOffset := 0);
FOR i := 0 TO 255 DO  str_temp[i] := 0; END_FOR
udiByteRead := sysfile.SysFileRead(hfile := hFile,pbyBuffer := ADR(str_temp), ulSize := 250, pResult := ADR(udiReadError));
str_temp := rm_return(str_temp);
IF udiByteRead > 7 THEN
	i_sTopicPublish := str_temp;
END_IF
sysfile.SysFileClose(hFile := hFile);	

hFile := sysfileopen(szFile := '/userapp/mqtt_topic_subscribe.txt', am := sysfile.AM_READ, pResult:= ADR(udiOpenError));
IF hFile = RTS_INVALID_HANDLE	THEN
	RETURN;
END_IF
 
//文件存在，开始读取内容
sysfile.SysFileSetPos(hFile:=hFile, ulOffset := 0);
FOR i := 0 TO 255 DO  str_temp[i] := 0; END_FOR
udiByteRead := sysfile.SysFileRead(hfile := hFile,pbyBuffer := ADR(str_temp), ulSize := 250, pResult := ADR(udiReadError));
str_temp := rm_return(str_temp);
IF udiByteRead > 7 THEN  
	i_sTopicSubscribe := str_temp;
END_IF
sysfile.SysFileClose(hFile := hFile);	

m_read_config := TRUE;
END_METHOD

END_FUNCTION_BLOCK

// Device/Application/MQTT_Client/Function Blocks/FB_CalculateRemainingLength
{attribute 'hide'}
FUNCTION_BLOCK FB_CalculateRemainingLength
VAR_INPUT
	wNumberOfBytes: WORD;
	
END_VAR
VAR_OUTPUT
	iNumberOfBytesRemianingLengthField: INT;
	arbyRemainingBytesField: ARRAY[0..3] OF BYTE;
END_VAR
VAR
	bEncodedByte: BYTE;
	wValue: WORD;
	iCount: INT;
END_VAR

wValue:=wNumberOfBytes;
iCount := 0;
REPEAT
	bEncodedByte:=UINT_TO_BYTE(wValue MOD 128);
	wValue:=wVALUE / 128;
	
	IF (wVALUE > 0) THEN
		bEncodedByte := (bEncodedByte AND 128);
	END_IF
	arbyRemainingBytesField[iCount] := bEncodedByte;
	iCount := iCount + 1;

UNTIL (wValue <= 0)
END_REPEAT;
iNumberOfBytesRemianingLengthField:=iCount;

END_FUNCTION_BLOCK

// Device/Application/MQTT_Client/Function Blocks/FB_Random
	{attribute 'hide'}
FUNCTION_BLOCK FB_Random
VAR_INPUT
	A: DWORD;
	B: DWORD;
	V: DWORD;
END_VAR
VAR_OUTPUT
	dwRandom: dword;
END_VAR
VAR
	dwValue1: DWORD;
	dwValue2: DWORD;
	M: DWORD;
	Q: DWORD;

END_VAR


Q:=Q+2;

M:=25;
dwRandom:=(A+V+B+Q) MOD M + 65;

END_FUNCTION_BLOCK

// Device/Application/MQTT_Client/Functions/MQTTPacket_len
FUNCTION MQTTPacket_len : CAA.SIZE
VAR_INPUT
	rem_len:INT;
END_VAR
VAR
END_VAR


rem_len := rem_len + 1; (* header byte *)

(* now remaining_length field *)
IF rem_len < 128 THEN
   rem_len := rem_len + 1;
ELSIF rem_len < 16384 THEN
   rem_len := rem_len + 2;
ELSIF rem_len < 2097151 THEN
   rem_len := rem_len + 3;
ELSE
   rem_len := rem_len + 4;
END_IF

MQTTPacket_len := rem_len;
RETURN;

END_FUNCTION

// Device/Application/MQTT_Client/Functions/MQTTPacket_encode
FUNCTION MQTTPacket_encode : INT
VAR_INPUT
	buf:POINTER TO BYTE;
	length : INT;
END_VAR
VAR
	rc : INT := 0;
	d : BYTE;
END_VAR


rc := 0;

WHILE length > 0  DO
	d := ANY_TO_BYTE(length MOD 128);
	length := length / 128;
	IF length > 0 THEN
		d := d + 16#80;
	END_IF
	buf[rc] := d;
	rc := rc + 1;
END_WHILE

MQTTPacket_encode := rc;

END_FUNCTION

// Device/Application/MQTT_Client/Functions/MQTT_connect_len
FUNCTION MQTT_connect_len : INT
VAR_INPUT
	len_clientId : INT;
	len_will_topic : INT;
	len_will_msg : INT;
	len_username : INT;
	len_password : INT;
END_VAR
VAR
	len :INT;
END_VAR


len := 10;  //  version 4

len := len + len_clientId + 2;

IF len_will_topic > 0 THEN
	len := len + len_will_topic + 2 + len_will_msg + 2;
END_IF

IF len_username > 0 THEN
	len := len + len_username + 2;
END_IF

IF len_password > 0 THEN
	len := len + len_password + 2;
END_IF


MQTT_connect_len := len;

END_FUNCTION

// Device/Application/MQTT_Client/Functions/json2arr
FUNCTION json2arr : INT
VAR_INPUT
	json : STRING(256);
	pArr : POINTER TO DUT_json;
	max_len : UINT;
END_VAR
VAR
	length : INT;  //length of json string
	number : INT;
	n : INT; 
	p :POINTER TO DUT_json;
	sj : STRING(255);
	str_val : STRING(255);
	
	kv:ARRAY[0..32] OF STRING(255);
	char_l : STRING(1);
	char_r : STRING(1);
	kv_str: STRING(255);
	pos : INT;
END_VAR

//将json格式的字符串分解为结构数组，当前支持的数据类型有： 整型、浮点型、字符串。 键值必须是字符串，并且不支持嵌套

json2arr := 0;

//check format
sj := json;
length := len(sj);
IF length < 7 THEN
	RETURN;
END_IF

n := count_char_in_string(sj, '{');
IF n <> 1 THEN
	RETURN;
END_IF

n := count_char_in_string(sj, '}');
IF n <> 1 THEN
	RETURN;
END_IF

n := count_char_in_string(sj, ',');

number := count_char_in_string(sj, ':');
IF number = 0 THEN
	RETURN;
END_IF

IF number - n <> 1 THEN  // ':'s are more 1 than ','
	RETURN;
END_IF

//split json to array of kv string
FOR n := 0 TO number - 1 DO
	char_l := ',';
	char_r := ',';
	IF n = 0 THEN
		char_l := '{';
	ELSIF n = number -1 THEN
		char_r := '}';
	END_IF
	kv[n] := get_sub_string(sj, char_l, char_r);
	sj := rm_left(sj, '"');  //remove '{' or ',' at the start of current string
	sj := rm_left(sj, char_r); //remove the first key-value
END_FOR

//split key and value, and move to recv_data which is pointed by pArr
FOR n := 0 TO number - 1 DO
	kv_str := kv[n];
	pos := find(kv_str, ':'); 
	IF  pos < 1 THEN  //error
		RETURN;
	END_IF
	
	pArr[n].key := get_sub_string(kv_str, '"', '"');
	str_val := get_sub_string(kv_str, ':', '&');

	IF find(str_val, '"') > 0 THEN //string
		pArr[n].val_tp := 2;
		pArr[n].value_str := get_sub_string(str_val, '"', '"');
	ELSIF find(str_val, '.') > 0 THEN //real
		pArr[n].val_tp := 1;
 		pArr[n].value_real := STRING_TO_REAL(str_val);
	ELSE
		pArr[n].val_tp := 0;
 		pArr[n].value_dint := STRING_TO_DINT(str_val);
	END_IF
		
END_FOR

json2arr := number;

END_FUNCTION

// Device/Application/MQTT_Client/Functions/count_char_in_string
FUNCTION count_char_in_string : int
VAR_INPUT
	in_str : STRING(255);
	ch : STRING(1);
END_VAR
VAR
	cnt : INT := 0;
	pos : INT;
	temp_str : STRING(255);
END_VAR



temp_str := in_str;

cnt := 0;
pos := find(temp_str, ch);
IF pos > 0 THEN
	cnt := cnt + 1;
END_IF

WHILE pos > 0 DO
	temp_str := right(temp_str, len(temp_str)-pos);
	pos := find(temp_str, ch);
	IF pos > 0 THEN
		cnt := cnt + 1;
	END_IF	
END_WHILE

count_char_in_string := cnt;

END_FUNCTION

// Device/Application/MQTT_Client/Functions/get_sub_string
FUNCTION get_sub_string : string(255)
VAR_INPUT
	in_str : STRING(255);
	char_l : STRING(1);
	char_r : STRING(1);
END_VAR
VAR
	start : INT;
	end : INT;
	sub_str : STRING(255);
	length : INT;
END_VAR

get_sub_string := '';

length := len(in_str);
start := 0;
end := length+1;

start := find(in_str, char_l);
sub_str := right(in_str, length-start);
length := len(sub_str);
end := find(sub_str, char_r);
IF end = 0 THEN
	end := length + 1;
END_IF
get_sub_string := left(sub_str, end-1);

END_FUNCTION

// Device/Application/MQTT_Client/Functions/rm_left
FUNCTION rm_left : string(255)
VAR_INPUT
	str_in:STRING(255);
	ch : string(1);
END_VAR
VAR
	pos : INT;
END_VAR


//删除字符串中特定字符左侧的部分，该字符保留。 如果没有发现该指定字符，则返回原字符串
rm_left := str_in;

pos := find(str_in, ch);
IF pos < 0 THEN
	RETURN; 
END_IF

rm_left := right(str_in, len(str_in)-pos+1);

END_FUNCTION

// Device/Application/MQTT_Client/Functions/arr2json_model
FUNCTION arr2json_model : STRING(255)
VAR_INPUT
	arr:ARRAY[0..32] OF dut_json;
	num : INT;
END_VAR
VAR
	i :INT;
	kv : DUT_json;
END_VAR


arr2json_model := '{"params":{';

FOR i := 0 TO num -1 DO
	kv := arr[i];
	arr2json_model := concat(arr2json_model, '"');
	arr2json_model := concat(arr2json_model, kv.key);
	arr2json_model := concat(arr2json_model, '":');
	IF kv.val_tp = GVL.TYPE_DINT THEN   
		arr2json_model := concat(arr2json_model, DINT_TO_STRING(kv.value_dint));		
	ELSIF kv.val_tp = GVL.TYPE_REAL THEN  
		arr2json_model := concat(arr2json_model, real2string(kv.value_real,2));
	ELSIF kv.val_tp = GVL.TYPE_STRING THEN  
		arr2json_model := concat(arr2json_model, '"');
		arr2json_model := concat(arr2json_model, kv.value_str);
		arr2json_model := concat(arr2json_model, '"');	
	ELSE
		arr2json_model := 'Error:  Value type is unknow.';
		RETURN;	
	END_IF
	IF i <> num-1 THEN
		arr2json_model := concat(arr2json_model, ',');
	END_IF
END_FOR

arr2json_model := concat(arr2json_model, '}}');

END_FUNCTION

// Device/Application/MQTT_Client/Functions/real2string
FUNCTION real2string : string
VAR_INPUT
	in:REAL;
	point:UINT := 2;  //小数点后的位数
END_VAR
VAR
	pp : INT; // point position
	ep : INT; // E position
	length:INT;
	str_org:STRING;
	E : UINT;
END_VAR

IF ABS(in) > 10000000 THEN
	real2string := DINT_TO_STRING(REAL_TO_DINT(in));
	RETURN;
END_IF

str_org := ANY_TO_STRING(in);
length := len(str_org);

pp := find(str_org, '.');
IF pp = 0 THEN //no ., the IN is integer
	real2string := str_org;
ELSIF length <= pp + point THEN // less than 2 
	real2string := str_org;
ELSE
	real2string := left(str_org, pp+point);
END_IF

RETURN;

// 处理科学计数法
ep := find(str_org, 'E');
IF ep = 0 THEN
	RETURN;
END_IF

// 超小浮点数 , 例如：  1.234553E-7
ep := find(str_org, 'E-');
IF ep > 0 THEN
	// 超小浮点数，尚待处理
    RETURN;
END_IF

// 超大浮点数，例如：  1.299993E09 ,保留整数部分
real2string := DINT_TO_STRING(REAL_TO_DINT(in));
RETURN;

END_FUNCTION

// Device/Application/MQTT_Client/Functions/real_arr2string
FUNCTION real_arr2string : STRING(256)
VAR_INPUT
	arr:ARRAY[0..19] OF REAL;
	num:DINT;
END_VAR
VAR
	i :DINT;
END_VAR

real_arr2string := '';

FOR i := 0 TO num-1 DO
	real_arr2string := concat(real_arr2string, real2string(arr[i],2));
	IF i <> num-1 THEN
		real_arr2string := concat(real_arr2string, ',');
	END_IF
END_FOR

END_FUNCTION

// Device/Application/gps/programs/prg_gps
PROGRAM prg_gps
VAR  
	filename:STRING(256) := '/tmp/connect_server.txt';
	hFile: RTS_IEC_HANDLE := 0;
	udiOpenError: RTS_IEC_RESULT;
	connect_open_flag :BOOL := TRUE;
	
	gps :Com_gps;
	com_handle :CAA.HANDLE; 
	packGPRMC : nmeaGPRMC;
	buf:STRING(255);
	gps_ok:BOOL := FALSE;
	
	in : REAL := 110.123456789;
	in2 : REAL;
	str_org :STRING(255);
	out : REAL;
	out2 : REAL;
	out3 : REAL;
	
	ind : LREAL := 110.123456789;
	in2d : LREAL;
	str_orgd :STRING(255);
	outd : LREAL;
	out2d : LREAL;
	out3d : LREAL;	
END_VAR

// just for test real to string
// in : REAL := 110.123456789;
in2 := in * 1000000;
str_org := real2string(in2,2);
out := STRING_TO_REAL(str_org);
out2  := in2 * 0.000001;
out3 := out2 * 1000000;

// double
// in : REAL := 110.123456789;
in2d := ind * 1000000;
str_orgd := real2string(in2d,2);
outd := STRING_TO_REAL(str_orgd);
out2d  := in2d * 0.000001;
out3d := out2d * 1000000;
// end of test



// 判断后端PPP网络是否连通，如果已经连通，则会同步网络时间
IF connect_open_flag THEN
	hFile := sysfileopen(szFile := filename, am := sysfile.AM_READ, pResult:= ADR(udiOpenError));
	IF hFile = RTS_INVALID_HANDLE THEN
		RETURN;
	END_IF
	
	hFile := MIC7001_BASE.close_file(hFile := hFile);
	connect_open_flag := FALSE;
END_IF

gps(xEnable := TRUE, com_hand := com_handle, gps_str => buf); 

nmea_parse_GPRMC(buf, SIZEOF(buf), ADR(packGPRMC));

IF packGPRMC.status = 'A' THEN
	gps_ok := TRUE;
ELSE
	gps_ok := FALSE;
END_IF

END_PROGRAM

// Device/Application/gps/functions/nmea_parse_GPRMC
FUNCTION nmea_parse_GPRMC : bool
VAR_INPUT
    buff : STRING(255);
	buff_sz : DINT;
	pack : POINTER TO nmeaGPRMC;
END_VAR
VAR
	str:STRING(255);
	rc :BOOL;
	checksum : DINT;	
END_VAR

nmea_parse_GPRMC := FALSE;

str := get_sub_string_1(buff, '$$', ',', 1);   //check 'GPRMC'
IF str <> 'GPRMC' THEN
	RETURN;
END_IF

//find time
str := get_sub_string_1(buff, ',', ',', 1);  
IF len(str) < len('hhmmss')  THEN
	RETURN;  //format error	
END_IF
IF NOT nmea_parse_time(str, ADR(pack^.utc)) THEN
	RETURN;
END_IF

//find status
str := get_sub_string_1(buff, ',', ',', 2);  
IF len(str)<1 THEN
	RETURN; //format error
END_IF
pack^.status := str;

//find lat
str := get_sub_string_1(buff, ',', ',', 3);  
IF len(str)<1 THEN
	RETURN; //format error
END_IF
pack^.lat := get_latlon_from_str(str);

//find ns
str := get_sub_string_1(buff, ',', ',', 4); 
IF len(str)<1 THEN
	RETURN; //format error
END_IF
pack^.ns := str;

//find lon
str := get_sub_string_1(buff, ',', ',', 5); 
IF len(str)<1 THEN
	RETURN; //format error
END_IF
pack^.lon := get_latlon_from_str(str);

//find ew
str := get_sub_string_1(buff, ',', ',', 6); 
IF len(str)<1 THEN
	RETURN; //format error
END_IF
pack^.ew := str;

//find speed
str := get_sub_string_1(buff, ',', ',', 7); 
IF len(str)<1 THEN
	RETURN; //format error
END_IF
pack^.speed := STRING_TO_REAL(str)*1.852;  // 节 -> km/h

//find direction
str := get_sub_string_1(buff, ',', ',', 8); 
IF len(str)<1 THEN
	RETURN; //format error
END_IF
pack^.direction := STRING_TO_REAL(str);

//find date
str := get_sub_string_1(buff, ',', ',', 9); 
IF len(str)<1 THEN
	RETURN; //format error
END_IF
IF NOT nmea_parse_date(str, ADR(pack^.utc)) THEN
	RETURN;
END_IF

//find declination
str := get_sub_string_1(buff, ',', ',', 10); 
IF len(str)<1 THEN
	pack^.declination := 0.0;
ELSE
	pack^.declination := STRING_TO_REAL(str);
END_IF

//find declin_ew
str := get_sub_string_1(buff, ',', ',', 11); 
IF len(str)<1 THEN
	RETURN; //format error
END_IF
pack^.declin_ew := str;

//find mode
str := get_sub_string_1(buff, ',', '*', 12); 
IF len(str) < 1 THEN
//	RETURN; // no mode is allowed
ELSE
	pack^.mode := str;
END_IF

//find checksum
str := get_sub_string_1(buff, '*', '$r', 1); 
IF len(str)<1 THEN
	RETURN; //format error
END_IF
checksum := STRING_TO_DINT(str);

nmea_parse_GPRMC := TRUE;

END_FUNCTION

// Device/Application/gps/functions/get_sub_string_1
FUNCTION get_sub_string_1 : STRING(255)
VAR_INPUT
	in_str : STRING(255);
	char_l : STRING(1);
	char_r : STRING(1);
	index : DINT := 1;
END_VAR
VAR
	start : DINT;
	end : DINT;
	sub_str : STRING(255);
	length : DINT;
	i :DINT;
END_VAR

get_sub_string_1 := '';
sub_str := in_str;
i := index;

length := len(sub_str);
start := 0;
end := length+1;

WHILE i > 0 DO
	start := find(sub_str, char_l);
	IF start = 0 THEN
		RETURN;
	END_IF
	sub_str := right(sub_str, DINT_TO_INT(length-start));
	length := len(sub_str);
	i := i - 1;
END_WHILE

end := find(sub_str, char_r);
IF end = 0 THEN
	end := length + 1;
END_IF
get_sub_string_1 := left(sub_str, DINT_TO_INT(end-1));

END_FUNCTION

// Device/Application/gps/functions/nmea_parse_time
FUNCTION nmea_parse_time : BOOL
VAR_INPUT
	str_time:STRING(255);
	p_utc:POINTER TO nmeaTIME;
END_VAR
VAR
	len_str:DINT;
END_VAR

nmea_parse_time := FALSE;

len_str := len(str_time);
IF len_str < len('hhmmss') THEN
	RETURN;  //format error
END_IF

p_utc^.hour := ANY_TO_DINT(left(str_time,2));
p_utc^.minute := ANY_TO_DINT(mid(str_time,2,3));
p_utc^.second := ANY_TO_DINT(mid(str_time,2,5));
IF len_str = len('hhmmss.u') THEN
	p_utc^.hsecond := ANY_TO_DINT(mid(str_time,1,8));
ELSIF len_str = len('hhmmss.uu') THEN
	p_utc^.hsecond := ANY_TO_DINT(mid(str_time,2,8));
ELSIF len_str = len('hhmmss.uuu') THEN
	p_utc^.hsecond := ANY_TO_DINT(mid(str_time,3,8));
ELSE
	//  no hsecond
END_IF

nmea_parse_time := TRUE;

END_FUNCTION

// Device/Application/gps/functions/get_latlon_from_str
FUNCTION get_latlon_from_str : REAL
VAR_INPUT
	str:STRING;
END_VAR

VAR
	temp:REAL;
	d:INT;
	m:REAL;
END_VAR

// lat format:   ddmm.mmmmmm  度度分分.分分分分分分
// lon format:  dddmm.mmmmmm  度度度分分.分分分分分分
   
temp := STRING_TO_REAL(str);
d := ANY_TO_INT(temp/100);
m := temp/100 - d;
m := m/0.6;

get_latlon_from_str := INT_TO_REAL(d)+m;

// 转换为：   度度度.度度度度度度

END_FUNCTION

// Device/Application/gps/functions/nmea_parse_date
FUNCTION nmea_parse_date : BOOL
VAR_INPUT
	str_time:STRING(255);
	p_utc:POINTER TO nmeaTIME;
END_VAR
VAR
	len_str:DINT;
END_VAR

nmea_parse_date := FALSE;

len_str := len(str_time);
IF len_str < len('ddmmyy') THEN
	RETURN;  //format error
END_IF

p_utc^.day := ANY_TO_DINT(left(str_time,2));
p_utc^.month := ANY_TO_DINT(mid(str_time,2,3));
p_utc^.year := ANY_TO_DINT(mid(str_time,2,5));

nmea_parse_date := TRUE;

END_FUNCTION

// Device/Application/gps/functionblocks/Com_gps
FUNCTION_BLOCK Com_gps
VAR_INPUT
	xEnable : BOOL := FALSE;
END_VAR
VAR_IN_OUT
	com_hand: CAA.HANDLE;
END_VAR
VAR_OUTPUT
	xDone : BOOL := FALSE;
	xError :BOOL := FALSE;
	xBusy : BOOL := FALSE;
	gps_str:STRING(255);
END_VAR
VAR
	ton_fb :TON;
	Com1Params: 			ARRAY [1..7] OF COM.PARAMETER;	(* Settings to communicate with 
the COM Port *)
	ComOpen: 				COM.Open;
	ComClose: 				COM.Close;
	ComWrite: 				COM.Write;
	ComRead: 				COM.Read;	
	Rcv_Cnt: 				CAA.SIZE;
	xCom1CloseError: 		BOOL;
	xCom1WriteError: 		BOOL;
	xCom1ReadError: 		BOOL;
	uiComState: INT := 0;
	ComID:USINT:=5;   //ttymxc4
	position :INT := 0;
	at_cmd :STRING := 'AT$r';
	at_buffer :STRING;
	ate0_cmd :STRING := 'ATE0$r';
	ate0_buffer :STRING;
	csq_cmd :STRING := 'AT+CSQ$r';
	csq_buffer :STRING;
	
	accid_cmd :STRING := 'AT+ICCID$r';
	iccid_read_buffer :STRING(255);
	ICCID_HEAD:STRING := '+ICCID: ';
	iccid:STRING(32);
	
	lac:STRING(4) := '0000';
	ci :STRING(4) := '0000';
	lac_set_cmd :STRING := 'AT+CREG=2$r';
	lac_read_cmd :STRING(255);
	
	
	lac_get_cmd :STRING := 'AT+CREG?$r';
	lac_read_buffer :STRING(255);
	
	lac_close_cmd :STRING := 'AT+CREG=0$r';
	lac_close_buffer :STRING(255);
	
	LACID_HEAD:STRING := '+CREG:';
	lac_str:STRING(8);
	ci_str:STRING(8);
	
	at_GPSCLOSE_buffer :STRING(255);
	at_GPSCLOSE_cmd :STRING := 'AT+QGPS=0$r';    
	at_GPSOPEN_cmd :STRING := 'AT+QGPS=1$r';     
	at_GPSOPEN_buffer :STRING(255);
	
	at_GPSSET_cmd :STRING := 'AT+QGPSCFG="nmeasrc",1$r';     
	at_GPSSET_buffer :STRING(255);
	
	at_GPSREAD_cmd :STRING := 'AT+QGPSGNMEA="RMC"$r';    
	at_GPSREAD_buffer :STRING(255);
	
	at_ask_buffer3 :STRING(1000);
	bit_start:INT;
	bit_end:INT;
	bit_start1:INT;
	bit_end1:INT;
	jd_info:STRING;
	wd_info:STRING;
	jd:REAL;
	wd:REAL;
	R_TIME:TIME;
	
	xDone_internal : BOOL := FALSE;
	xError_internal :BOOL := FALSE;
	
	sudu_info :STRING;
	bit_end2:INT;
	sd:REAL;
	
	ton_err:ton;
	cntr_40:DINT := 0;
END_VAR

IF NOT xEnable THEN
	xDone := FALSE;
	xError := FALSE;
	xBusy := FALSE;
	uiComState := 0;
	RETURN;
END_IF

CASE uiComState OF
	0:
	Com1Params[1].udiParameterId := COM.CAA_Parameter_Constants.udiPort;
	Com1Params[1].udiValue := ComID; 
	Com1Params[2].udiParameterId := COM.CAA_Parameter_Constants.udiBaudrate;
	Com1Params[2].udiValue := 115200;
	Com1Params[3].udiParameterId := COM.CAA_Parameter_Constants.udiParity;
	Com1Params[3].udiValue := INT_TO_UINT(COM.PARITY.NONE);
	Com1Params[4].udiParameterId := COM.CAA_Parameter_Constants.udiStopBits;
	Com1Params[4].udiValue := INT_TO_UINT(COM.STOPBIT.ONESTOPBIT);
	Com1Params[5].udiParameterId := COM.CAA_Parameter_Constants.udiTimeout;
	Com1Params[5].udiValue := 0;
	Com1Params[6].udiParameterId := COM.CAA_Parameter_Constants.udiByteSize;
	Com1Params[6].udiValue := 8;
	Com1Params[7].udiParameterId := COM.CAA_Parameter_Constants.udiBinary;
	Com1Params[7].udiValue := 0;					
	ComOpen(xExecute := TRUE, usiListLength:=UINT_TO_USINT(SIZEOF(Com1Params)/SIZEOF(COM.PARAMETER)),pParameterList:= ADR(Com1Params),hCom=> com_hand);			
	IF ComOpen.xError THEN
		ton_err(in := FALSE, pt := T#5S);
		uiComState := 32767;
	ELSIF ComOpen.xDone THEN
		uiComState := 1;
		com_hand := ComOpen.hCom;
		ComWrite(xExecute := FALSE,hCom:= com_hand);	
		ComRead(xExecute := FALSE,hCom:= com_hand);
	END_IF
	
	1:  // write "AT\r"
	ComWrite(xExecute := TRUE,hCom:= com_hand,pBuffer:= ADR(at_cmd),szSize:=len(at_cmd));		
	IF ComWrite.xError THEN
		uiComState := 200;
	END_IF
	IF ComWrite.xDone THEN
		ComWrite(xExecute := FALSE, hCom:= com_hand);
		uiComState := 2;
	END_IF
	
	2:
	ton_fb(IN := TRUE, PT := TIME#300MS);
	IF (ton_fb.Q) THEN
		ton_fb(IN := FALSE, PT := TIME#300MS);
		uiComState := 3;
	END_IF
	
	3:
	ComRead(xExecute := TRUE,hCom:= com_hand, pBuffer:= ADR(at_buffer), szBuffer:= SIZEOF(at_buffer));			
	IF ComRead.xError THEN
		uiComState := 32767;
	END_IF
	IF ComRead.xDone THEN
		position := find(at_buffer, 'OK');
		IF position > 0 THEN
			uiComState := 10;
		ELSE
			uiComState := 200;
		END_IF
		ComRead(xExecute := FALSE, hCom:= com_hand);
	END_IF
	
(*	
	4: // write "ATE0\r"
	ComWrite(xExecute := TRUE,hCom:= com_hand,pBuffer:= ADR(ate0_cmd),szSize:=len(ate0_cmd));		
	IF ComWrite.xError THEN
		uiComState := 200;
	END_IF
	IF ComWrite.xDone THEN
		ComWrite(xExecute := FALSE, hCom:= com_hand);
		uiComState := 5;
	END_IF
	
	5:
	ton_fb(IN := TRUE, PT := TIME#300MS);
	IF (ton_fb.Q) THEN
		ton_fb(IN := FALSE, PT := TIME#300MS);
		uiComState := 6;
	END_IF
	
	6:
	ComRead(xExecute := TRUE,hCom:= com_hand, pBuffer:= ADR(ate0_buffer), szBuffer:= SIZEOF(ate0_buffer));			
	IF ComRead.xError THEN
		uiComState := 200;
	END_IF
	IF ComRead.xDone THEN
		position := find(ate0_buffer, 'OK');
		IF position > 0 THEN
			uiComState := 10;
		ELSE
			uiComState := 200;
		END_IF
		ComRead(xExecute := FALSE, hCom:= com_hand);
	END_IF
	*)
	
	
	10: // write "AT+CSQ\r"
	ComWrite(xExecute := TRUE,hCom:= com_hand,pBuffer:= ADR(csq_cmd),szSize:=len(csq_cmd));		
	IF ComWrite.xError THEN
		uiComState := 200;
	END_IF
	IF ComWrite.xDone THEN
		ComWrite(xExecute := FALSE, hCom:= com_hand);
		uiComState := 11;
	END_IF
	
	11:
	ton_fb(IN := TRUE, PT := TIME#300MS);
	IF (ton_fb.Q) THEN
		ton_fb(IN := FALSE, PT := TIME#300MS);
		uiComState := 12;
	END_IF
	
	12:
	ComRead(xExecute := TRUE,hCom:= com_hand, pBuffer:= ADR(csq_buffer), szBuffer:= SIZEOF(csq_buffer));			
	IF ComRead.xError THEN
		uiComState := 200;
	END_IF
	IF ComRead.xDone THEN
		position := find(csq_buffer, 'OK');
		IF position > 0 THEN
			uiComState := 13;
		ELSE
			uiComState := 200;
		END_IF
		ComRead(xExecute := FALSE, hCom:= com_hand);
	END_IF
	
	13:
	ComWrite(xExecute := TRUE,hCom:= com_hand,pBuffer:= ADR(accid_cmd),szSize:=len(accid_cmd));		
	IF ComWrite.xError THEN
		uiComState := 200;
	END_IF
	IF ComWrite.xDone THEN
		ComWrite(xExecute := FALSE, hCom:= com_hand);
		uiComState := 14;
	END_IF
	
	14:
	ton_fb(IN := TRUE, PT := TIME#300MS);
	IF (ton_fb.Q) THEN
		ton_fb(IN := FALSE, PT := TIME#300MS);
		uiComState := 15;
	END_IF
	
	15:
	ComRead(xExecute := TRUE,hCom:= com_hand, pBuffer:= ADR(iccid_read_buffer), szBuffer:= SIZEOF(iccid_read_buffer));			
	IF ComRead.xError THEN
		uiComState := 200;
	END_IF
	IF ComRead.xDone THEN
		IF ComRead.szsize > 0 THEN
			position := find(iccid_read_buffer, ICCID_HEAD);
			IF position > 0 THEN
				iccid := mid(iccid_read_buffer, 20, position + len(ICCID_HEAD));
				uiComState := 16;
			ELSE
				uiComState := 200;
			END_IF
		ELSE
			uiComState := 200;
		END_IF
		ComRead(xExecute := FALSE, hCom:= com_hand);
	END_IF
	
	16:
	ComWrite(xExecute := TRUE,hCom:= com_hand,pBuffer:= ADR(at_GPSCLOSE_cmd),szSize:=len(at_GPSCLOSE_cmd));		
	IF ComWrite.xError THEN
		uiComState := 200;
	END_IF
	IF ComWrite.xDone THEN
		ComWrite(xExecute := FALSE, hCom:= com_hand);
		uiComState := 17;
	END_IF
	
	17:
	ton_fb(IN := TRUE, PT := TIME#300MS);
	IF (ton_fb.Q) THEN
		ton_fb(IN := FALSE, PT := TIME#300MS);
		uiComState := 18;
	END_IF
	
	18:
	ComRead(xExecute := TRUE,hCom:= com_hand, pBuffer:= ADR(at_GPSCLOSE_buffer), szBuffer:= SIZEOF(at_GPSCLOSE_buffer));			
	IF ComRead.xError THEN
		uiComState := 200;
	END_IF
	IF ComRead.xDone THEN
		uiComState := 25;
		ComRead(xExecute := FALSE, hCom:= com_hand);
	END_IF
	
	25:
	ComWrite(xExecute := TRUE,hCom:= com_hand,pBuffer:= ADR(at_GPSOPEN_cmd),szSize:= len(at_GPSOPEN_cmd));		
	IF ComWrite.xError THEN
		uiComState := 200;
	END_IF
	IF ComWrite.xDone THEN		
		ComWrite(xExecute := FALSE);
		uiComState := 26;
	END_IF
	
	26:
	ton_fb(IN := TRUE, PT := TIME#300MS);
	IF (ton_fb.Q) THEN
		ton_fb(IN := FALSE, PT := TIME#300MS);
		uiComState := 27;
	END_IF

	27:
	ComRead(xExecute := TRUE,hCom:= com_hand, pBuffer:= ADR(at_GPSOPEN_buffer), szBuffer:= SIZEOF(at_GPSOPEN_buffer));			
	IF ComRead.xError THEN
		uiComState := 200;
	END_IF
	IF ComRead.xDone THEN
		position := find(at_GPSOPEN_buffer, 'OK');
		IF position > 0 THEN
			uiComState := 28;
		ELSE
			uiComState := 200;
		END_IF
		ComRead(xExecute := FALSE, hCom:= com_hand);
	END_IF
	
	
	28:
	ComWrite(xExecute := TRUE,hCom:= com_hand,pBuffer:= ADR(at_GPSSET_cmd),szSize:= len(at_GPSSET_cmd));		//发送AT指令，查询获取的经纬度
	IF ComWrite.xError THEN
		uiComState := 200;
	END_IF
	IF ComWrite.xDone THEN		
		ComWrite(xExecute := FALSE);
		uiComState := 29;
	END_IF
	
	29:
	ton_fb(IN := TRUE, PT := TIME#300MS);
	IF (ton_fb.Q) THEN
		ton_fb(IN := FALSE, PT := TIME#300MS);
		uiComState := 30;
	END_IF
	
	30:
	ComRead(xExecute := TRUE,hCom:= com_hand, pBuffer:= ADR(at_GPSSET_buffer), szBuffer:= SIZEOF(at_GPSSET_buffer));			
	IF ComRead.xError THEN
		uiComState := 200;
	END_IF
	IF ComRead.xDone THEN
		position := find(at_GPSSET_buffer, 'OK');
		IF position > 0 THEN
			uiComState := 31;
		ELSE
			uiComState := 200;
		END_IF
		ComRead(xExecute := FALSE, hCom:= com_hand);
	END_IF
	
	
	31:
	ComWrite(xExecute := TRUE,hCom:= com_hand,pBuffer:= ADR(at_GPSREAD_cmd),szSize:= len(at_GPSREAD_cmd));		//发送AT指令，查询获取的经纬度
	IF ComWrite.xError THEN
		uiComState := 200;
	END_IF
	IF ComWrite.xDone THEN		
		ComWrite(xExecute := FALSE);
		uiComState := 32;
	END_IF

	32:
	ton_fb(IN := TRUE, PT := TIME#300MS);
	IF (ton_fb.Q) THEN
		ton_fb(IN := FALSE, PT := TIME#300MS);
		uiComState := 33;
	END_IF
	
	33:
	ComRead(xExecute := TRUE,hCom:= com_hand, pBuffer:= ADR(at_GPSREAD_buffer), szBuffer:= SIZEOF(at_GPSREAD_buffer));
	IF ComRead.xError THEN
		uiComState := 200;
	END_IF
    IF ComRead.xDone THEN
		gps_str := at_GPSREAD_buffer;
		uiComState := 40;
		cntr_40 := 0;
		ComRead(xExecute := FALSE, hCom:= com_hand);
	END_IF
	
	40:  // waiting
	   cntr_40 := cntr_40+1;
	   IF cntr_40 > 20 THEN // 2s
		   uiComState := 31;
	   END_IF
	
	200:
		xError_internal := TRUE;
		uiComState := 202;
		
	201:
		xDone_internal := TRUE;
		uiComState := 202;
		
	202:
		ComClose(xExecute := FALSE, hCom:= com_hand); 	
		uiComState := 203;
	
	203:
		ComClose(xExecute := TRUE,hCom:= com_hand);
		IF ComClose.xError THEN
			uiComState := 32767;
		END_IF
		
		IF ComClose.xDone THEN
			ComClose(xExecute := FALSE, hCom:= com_hand); 	
		
			IF xDone_internal THEN
				uiComState := 255;
			END_IF
			
			IF xError_internal THEN
				uiComState := 32767;
			END_IF
		END_IF
	
	
	255:
		xDone := TRUE;
		
	32767:	
		xError := TRUE;
		ton_err(in := TRUE, pt := T#5S);
		IF ton_err.Q THEN
			ComOpen(xExecute := FALSE, usiListLength:=UINT_TO_USINT(SIZEOF(Com1Params)/SIZEOF(COM.PARAMETER)),pParameterList:= ADR(Com1Params),hCom=> com_hand);	
			ton_err(in := FALSE, pt := T#5S);
			uiComState := 0;
		END_IF
END_CASE

END_FUNCTION_BLOCK

// Device/Application/prg_jt808
PROGRAM prg_jt808
VAR
	inited : BOOL := FALSE;
	fluidLow:INT := 0;
	lossWater:INT := 0;
	dirtyWater:INT := 0;
	littleWater:INT := 0;
	pressSuper:INT := 0;
	
	strShmFileDown : STRING := 'SHM_JT808_DW_7001';
	strShmFileUp : STRING := 'SHM_JT808_UP_7001';
	hShMemDown: RTS_IEC_HANDLE := RTS_INVALID_HANDLE ;
	hShMemUp: RTS_IEC_HANDLE := RTS_INVALID_HANDLE ;
	ResultRead: RTS_IEC_RESULT;
	ResultWrite: RTS_IEC_RESULT;
	
	iRead: __UXINT;
	iWrite: __UXINT;
	shmDataDown:stShmJT808Down;
	shmDataUp:stShmJT808Up;
	sizeOfStFromAliyun:__UXINT := SIZEOF(stShmJT808Down);
	sizeOfStToAliyun:__UXINT := SIZEOF(stShmJT808Up);
	
	sim_data : DINT := 0;
	digi_val :DWORD := 0;
	lock_1 :BOOL := FALSE;
	lock_2 :BOOL := FALSE;
	unlock :BOOL := FALSE;
	test_val2 :DINT;
	
	get_dt:dtu.GetDateandTime();
	tempdt : DWORD;
	g_uiYear:UINT;
	g_uiMonth:UINT;
	g_uiDate:UINT;
	g_uiHour:UINT;
	g_uiMinute:UINT;
	g_uiSecond:UINT;
END_VAR


IF NOT inited THEN
 	IF NOT init_shm() THEN  // 初始化失败
		RETURN;
	ELSE
		inited := TRUE;
		
		sim_data := 0;
		test_val2 := 0;
	END_IF  
END_IF

IF read_from_server() THEN
   // 读取服务器发来的数据
	IF shmDataDown.ctrl > 0 THEN
		// 处理命令通道1
	END_IF
END_IF

// 准备上传到服务器的数据
sim_data := sim_data + 1;

get_dt(xExecute := TRUE);
 IF get_dt.xDone THEN
  tempdt := DT_TO_DWORD(get_dt.dtDateandtime);
  tempdt := tempdt + 3600*8;   // utc 时间转为北京时间
  dtu.DTSplit(DWORD_TO_DT(tempdt), ADR(g_uiYear), ADR(g_uiMonth), ADR(g_uiDate), ADR(g_uiHour), ADR(g_uiMinute), ADR(g_uiSecond));

  get_dt(xExecute := FALSE);

 END_IF

shmDataUp.location.asc_time[0] := ANY_TO_BYTE(g_uiYear MOD 100);
shmDataUp.location.asc_time[1] := ANY_TO_BYTE(g_uiMonth);
shmDataUp.location.asc_time[2] := ANY_TO_BYTE(g_uiDate);
shmDataUp.location.asc_time[3] := ANY_TO_BYTE(g_uiHour);
shmDataUp.location.asc_time[4] := ANY_TO_BYTE(g_uiMinute);
shmDataUp.location.asc_time[5] := ANY_TO_BYTE(g_uiSecond);
(*
shmDataUp.loc_ext.km_all := ANY_TO_DINT( gvl_es.trip_all_1939*10);      // jt808 unit: 0.1Km
shmDataUp.loc_ext.fuel_trip := ANY_TO_DINT(gvl_es.fuel_trip_engine*2);  // jt808 unit: 0.5L
shmDataUp.loc_ext.fuel_all := ANY_TO_DINT( gvl_es.fuelall_engine*2);    // jt808 unit: 0.5L
shmDataUp.loc_ext.fuel_r_h := ANY_TO_DINT(gvl_es.fuelrate_engine*20);   // jt808 unit: 0.05L/h
IF gvl_es.fuel_100km = 0 OR gvl_es.fuel_100km = 999 THEN
	shmDataUp.loc_ext.fuel_r_l := 0;
ELSE
	shmDataUp.loc_ext.fuel_r_l := ANY_TO_DINT(512*100/gvl_es.fuel_100km);   // jt808 unit: 1/512Km/L
END_IF
*)

IF prg_gps.packGPRMC.status = 'A' THEN  // GPS定位成功
	shmDataUp.location.latitude := ANY_TO_DINT(prg_gps.packGPRMC.lat*1000000);
	shmDataUp.location.longitude := ANY_TO_DINT(prg_gps.packGPRMC.lon*1000000);
	shmDataUp.location.altitude := 54;
	shmDataUp.location.speed := ANY_TO_INT(prg_gps.packGPRMC.speed);
	shmDataUp.location.bearing := ANY_TO_INT(prg_gps.packGPRMC.direction);
	shmDataUp.location.status := 16#03;   
ELSIF 	prg_gps.packGPRMC.status = 'V' THEN  // 有GPS，但尚未定位成功
	shmDataUp.location.latitude := 0;
	shmDataUp.location.longitude := 0;	
	shmDataUp.location.altitude := 0;
	shmDataUp.location.speed := 0;
	shmDataUp.location.bearing := 0;	
	shmDataUp.location.status := 16#02;   
ELSE	// 没有GPS
    shmDataUp.loc_ext.lac := MIC7001_base.read_num_from_file(filename := '/tmp/lac.txt');
	shmDataUp.loc_ext.cid := MIC7001_base.read_num_from_file(filename := '/tmp/cid.txt');
	shmDataUp.location.latitude := 28230306;
	shmDataUp.location.longitude := 113414176;	
	shmDataUp.location.altitude := 0;	
	shmDataUp.location.status := 16#03;   
END_IF

IF send_to_server() THEN
	// write ok
END_IF

METHOD send_to_server : bool
VAR_INPUT
END_VAR
send_to_server := FALSE;

iWrite := sysshm.SysSharedMemoryWrite(hShMemUp, 0, ADR(shmDataUp), sizeOfStToAliyun, ADR(ResultWrite));
IF iWrite = sizeOfStToAliyun THEN
	send_to_server := TRUE;
END_IF

RETURN;
END_METHOD

METHOD read_from_server : bool
VAR_INPUT
END_VAR
read_from_server := FALSE;

iRead := sysshm.SysSharedMemoryRead(hShMemDown, 0, ADR(shmDataDown), sizeOfStFromAliyun, ADR(ResultRead));
IF iRead = sizeOfStFromAliyun THEN
    read_from_server := TRUE;
END_IF

RETURN;
END_METHOD

METHOD init_shm : bool
VAR_INPUT
END_VAR
init_shm := FALSE;

IF hShMemDown = RTS_INVALID_HANDLE  THEN
	hShMemDown := sysshm.SysSharedMemoryCreate(strShmFileDown, 0, ADR(sizeOfStFromAliyun), ADR(ResultRead));	
END_IF

IF hShMemUp = RTS_INVALID_HANDLE  THEN
	hShMemUp := sysshm.SysSharedMemoryCreate(strShmFileUp, 0, ADR(sizeOfStToAliyun), ADR(ResultRead));	
END_IF

IF hShMemDown = RTS_INVALID_HANDLE  OR hShMemUp = RTS_INVALID_HANDLE  THEN
	RETURN;
END_IF

init_shm := TRUE;
RETURN;
END_METHOD

END_PROGRAM

// Device/Application/MQTT_Client/Function Blocks/FB_DecodeRemainingLength
FUNCTION_BLOCK FB_DecodeRemainingLength
VAR_INPUT
	abyRemainingLengthField: ARRAY[0..3] OF BYTE;
END_VAR
VAR_OUTPUT
	uiRemeiningLength: UINT;
END_VAR
VAR
	multiplier: UINT;
	value: UINT;
	iCount: INT;
END_VAR

multiplier := 1;
value := 0;
iCount :=0;
REPEAT
	value := value + (abyRemainingLengthField [iCount] AND 127)*multiplier;
	multiplier := multiplier * 128;
UNTIL ((abyRemainingLengthField [iCount] AND 128) <> 0)
END_REPEAT;
uiRemeiningLength:=value;

END_FUNCTION_BLOCK
